# EPICS substitutions: apps/dcPowerApp/Db/magflow.substitutions
file "db/magflow.db" {
    pattern { P R CH PORT ASLO EGU }
    { B_SOL:   MPS:ret_   1 L2 0.01 gpm }
    { B_TORUS: MPS:fsw1:   2 L2 0.01 lpm }
    { B_TORUS: MPS:fsw2:   3 L2 0.01 lpm }
    { B_TORUS: MPS:fsw3:   4 L2 0.01 lpm }
    { B_TORUS: MPS:fsw4:   5 L2 0.01 lpm }
    { B_TORUS: MPS:fsw5:   6 L2 0.01 lpm }
}
